// TIA Portal V20 export
// export: Created 2025-12-01T14:57:28.059015Z, ExportSetting None, DisplayName Totally Integrated Automation Portal, DisplayVersion V20 Update 3, DisplayName TIA Portal Openness, DisplayVersion V20 Update 3, DisplayName TIA Portal Version Control Interface, DisplayVersion V20 Update 3, DisplayName STEP 7 Professional, DisplayVersion V20 Update 3, DisplayName STEP 7 Safety, DisplayVersion V20 Update 2, DisplayName WinCC Basic/Comfort/Advanced, DisplayVersion V20 Update 3, DisplayName WinCC Professional, DisplayVersion V20 Update 3, DisplayName WinCC Unified, DisplayVersion V20 Update 3
FUNCTION_BLOCK "FB601_EntradaFija_Quimarox"   // FB601, LAD
{ S7_Optimized_Access := 'FALSE' }
// stored: AutoNumber false, SetENOAutomatically false
   VAR_INPUT
      MesaAnterior : UInt;
      MesaDeCarga : UInt;
      ID_Quimarox : UInt;
      ID_Elemento : UInt;
      EnTension : Bool;
      Termico : Bool;
      pHs_PosicionCarga : Bool;
      pHs_Protrusion : Bool;
      PRV_AVTF : Bool;
      PRV_DescargaActiva : Bool;
      V_FILTRO_pHsPresencia : Int;
      Pto_Ajuste_1 : Int;
   END_VAR
   VAR_OUTPUT
      PRV_PTF : Bool;   // permiso mesa anterior y avance de la siguiente
      PRV_FTF : Bool;
      PararElevador : Bool;
      ElevadorEnLenta : Bool;
      Avance_EntradaFija : Bool;
   END_VAR
   VAR_IN_OUT
      ROUTING_Destino : UInt;
      ROUTING_Etiqueta : UDInt;
   END_VAR
   VAR
      TMP_EnTension { S7_SetPoint := 'True'} : "FB910_CNT_UHS";
      FILTRO_pHsPresencia { S7_SetPoint := 'True'} : "FB910_CNT_UHS";
      EstadoAsociadoEnMesa : UInt;
      Aux_PeineDeCarga : UInt;
      PresenciaEnReset : Bool;
   END_VAR
   VAR_TEMP
      TMP_PeineDeCarga : UInt;
      TMP_PeineLiberar : UInt;
      MesaQuimarox : UInt;
      VagonReservado : UInt;
      NumeroUT : UInt;
      EsMesaTL : Bool;
      FILTRO_PosicionCarga : Bool;
   END_VAR
BEGIN

NETWORK
TITLE = ERROR - Rearme
/////////////////////////////////////////////////////////////
/////////////////////////////////////////////////////////////
/////////////////////////////////////////////////////////////
// Rearne de Errores
      SET;
      A     "DB902_Estado_ZonaMesa".EstadoMesas[#MesaDeCarga].Rearme_CBx;
      O     "DB902_Estado_ZonaMesa".EstadoMesas[#MesaDeCarga].PerReset_CBx;
      R     "DB900_Estado_Mesas".EstadoVI[#MesaDeCarga].Error_Mx;
      R     "DB900_Estado_Mesas".EstadoVI[#MesaDeCarga].Err_Protusion;
      R     "DB900_Estado_Mesas".EstadoVI[#MesaDeCarga].Err_TOut_Avance_E1_E3;
      R     "DB900_Estado_Mesas".EstadoVI[#MesaDeCarga].Err_DatosPLC;
      R     "DB900_Estado_Mesas".EstadoVI[#MesaDeCarga].Err_Termico_E1_E3;



NETWORK
TITLE = RECEP OK DE LA ORDEN -- NO SE UTILIZA
/////////////////////////////////////////////////////////////
/////////////////////////////////////////////////////////////
/////////////////////////////////////////////////////////////
// RECEP OK DE LA ORDEN
      SET;
      AN    "DB841_Recepcion".Mesa[#MesaDeCarga].Protocolo.Ord_S00;
      AN    "DB841_Recepcion".Mesa[#MesaDeCarga].Protocolo.Ord_S01;
      AN    "DB841_Recepcion".Mesa[#MesaDeCarga].Protocolo.Ord_S02;
      AN    "DB841_Recepcion".Mesa[#MesaDeCarga].Protocolo.Ord_S03;
      NOT;
      =     "DB840_Emision".Mesa[#MesaDeCarga].Protocolo.RecepOK;



NETWORK
TITLE = HMI - Manual
/////////////////////////////////////////////////////////////
/////////////////////////////////////////////////////////////
/////////////////////////////////////////////////////////////
// Para HMI >>> Manual
      SET;
      O     "DB902_Estado_ZonaMesa".EstadoMesas[#MesaDeCarga].Manual_CBx;
      =     "DB900_Estado_Mesas".EstadoVI[#MesaDeCarga].Manual;



NETWORK
TITLE = HMI - Entradas y Salidas de la Mesa
/////////////////////////////////////////////////////////////
/////////////////////////////////////////////////////////////
/////////////////////////////////////////////////////////////
// Entradas
      SET;
      A     #pHs_PosicionCarga;
      =     "DB900_Estado_Mesas".EstadoVI[#MesaDeCarga].En_PHS_1;
      SET;
      A     #pHs_Protrusion;
      =     "DB900_Estado_Mesas".EstadoVI[#MesaDeCarga].En_pHs_Prot1;

      SET;
      A     #Termico;
      =     "DB900_Estado_Mesas".EstadoVI[#MesaDeCarga].En_Termico1;

// Salidas
      SET;
      A     #Avance_EntradaFija;
      =     "DB900_Estado_Mesas".EstadoVI[#MesaDeCarga].Sa_Rod_Avance;



NETWORK
TITLE = Comprobacion de que la MESA es de TRACKING
/////////////////////////////////////////////////////////////
/////////////////////////////////////////////////////////////
/////////////////////////////////////////////////////////////
// Comprobar si es una Mesa de Tracking o Routing
      SET;
      A     "DB850_DefinicionMesas".Mesa[#MesaDeCarga].ConfigMesa.MesaTL;
      =     #EsMesaTL;



REGION Network 6: TMP - Espera En Tension
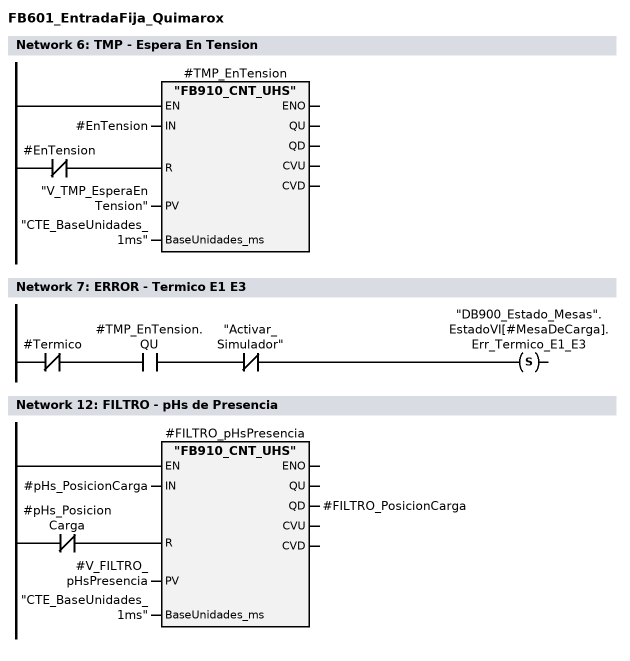
   RUNG wire#powerrail
      #TMP_EnTension(R := wire#w1, IN := #EnTension, PV := "V_TMP_EsperaEnTension", BaseUnidades_ms := "CTE_BaseUnidades_1ms", QU =>, QD =>, CVU =>, CVD =>)
   END_RUNG
   RUNG wire#powerrail
      I_Contact( #EnTension )
   END_RUNG wire#w1
   // the same network as SCL:
   #TMP_EnTension(IN := #EnTension,   // "FB910_CNT_UHS"
                  R := NOT #EnTension,
                  PV := "V_TMP_EsperaEnTension",
                  BaseUnidades_ms := "CTE_BaseUnidades_1ms");
END_REGION

REGION Network 7: ERROR - Termico E1 E3
   RUNG wire#powerrail
      I_Contact( #Termico )
      Contact( #TMP_EnTension.QU )
      I_Contact( "Activar_Simulador" )
      S_Coil( "DB900_Estado_Mesas".EstadoVI[#MesaDeCarga].Err_Termico_E1_E3 )
   END_RUNG
   // the same network as SCL:
   IF NOT #Termico AND #TMP_EnTension.QU AND NOT "Activar_Simulador" THEN
       "DB900_Estado_Mesas".EstadoVI[#MesaDeCarga].Err_Termico_E1_E3 := TRUE;
   END_IF;
END_REGION

NETWORK
TITLE = INICIALIZACION Previa
/////////////////////////////////////////////////////////////
/////////////////////////////////////////////////////////////
/////////////////////////////////////////////////////////////
      CLR;
      =     #PRV_PTF;
      =     #PRV_FTF;

      CLR;
      =     #ElevadorEnLenta;
      =     #PararElevador;
      =     #Avance_EntradaFija;

      CLR;
      =     "DB900_Estado_Mesas".EstadoVI[#MesaDeCarga].Etapas_Reset;
      =     "DB900_Estado_Mesas".EstadoVI[#MesaDeCarga].Etapa_Vacia;
      =     "DB900_Estado_Mesas".EstadoVI[#MesaDeCarga].Etapa_Cargada;
      =     "DB900_Estado_Mesas".EstadoVI[#MesaDeCarga].Etapas_Carga_E1;
      =     "DB900_Estado_Mesas".EstadoVI[#MesaDeCarga].Etapas_Descarga_S0;



NETWORK
TITLE = SISTEMA - Paro Blando
/////////////////////////////////////////////////////////////
/////////////////////////////////////////////////////////////
/////////////////////////////////////////////////////////////
// - Inicializar Variables de PARO BLANDO
      CLR;
      =     "DB900_Estado_Mesas".EstadoVI[#MesaDeCarga].Paro_Blando;

/////////////////////////////////////////////////////////////
// - Existe PARO BLANDO ???
      SET;
      AN    "DB902_Estado_ZonaMesa".EstadoMesas[#MesaDeCarga].ParoBlando_CBx;
      JC    NoRealizandose_ParoBlando;

/////////////////////////////////////////////////////////////
// - Fin de PARO BLANDO
      SET;
      =     "DB900_Estado_Mesas".EstadoVI[#MesaDeCarga].Paro_Blando;


/////////////////////////////////////////////////////////////
/////////////////////////////////////////////////////////////
/////////////////////////////////////////////////////////////
// - Final Tratamiento del PARO BLANDO
NoRealizandose_ParoBlando:NOP   0;



NETWORK
TITLE = SISTEMA - Reset
/////////////////////////////////////////////////////////////
/////////////////////////////////////////////////////////////
/////////////////////////////////////////////////////////////
// -- Inicializar Variables de RESET
      SET;
      AN    "DB902_Estado_ZonaMesa".EstadoMesas[#MesaDeCarga].PerReset_CBx;
      R     "DB900_Estado_Mesas".EstadoVI[#MesaDeCarga].Fin_VI;
      R     #PresenciaEnReset;

/////////////////////////////////////////////////////////////
/////////////////////////////////////////////////////////////
/////////////////////////////////////////////////////////////
// - Existe RESET ??
      SET;
      AN    "DB902_Estado_ZonaMesa".EstadoMesas[#MesaDeCarga].PerReset_CBx;
      JC    NoRealizandose_Reset;

      L     0;  // Estado de La Mesa = 0
      T     #EstadoAsociadoEnMesa;
      SET;
      =     "DB900_Estado_Mesas".EstadoVI[#MesaDeCarga].Etapas_Reset;

/////////////////////////////////////////////////////////////
/////////////////////////////////////////////////////////////
/////////////////////////////////////////////////////////////
// - Emision de Presencia en caso de Reset
      SET;  // Presencia >>> Reset Total
      A     #pHs_PosicionCarga;
      A     "DB831_Mesas".Mesas[#MesaDeCarga].Memorias.M_ResetTotal;
      AN    #PresenciaEnReset;
      JC    Enviar_PresenciaEnResetTotal;

      SET;  // Presencia >>> Reset Parcial
      A     #pHs_PosicionCarga;
      A     "DB831_Mesas".Mesas[#MesaDeCarga].Memorias.M_ResetParcial;
      AN    #PresenciaEnReset;
      JC    Enviar_PresenciaEnResetParcial;

      JU    Final_PresenciaEnReset;

// - Presencia en Reset TOTAL >>> Enviar NUUT
Enviar_PresenciaEnResetTotal:NOP   0;
      CALL  "FC723_InsertarUT_EnMesa"
      ( MesaActual := #MesaDeCarga,
        NumeroUT   := #NumeroUT
      );
      L     132;  // Envio de Nueva UT en RESET
      T     "DB812_UTs_Control".UT[#NumeroUT].EstadoEventoAGenerar;

      SET;  // Ya esta Avisado el JdT
      S     #PresenciaEnReset;

      JU    Final_PresenciaEnReset;

// - Presencia en Reset Parcial >>> Enviar LOCA en Reset Pantalla
Enviar_PresenciaEnResetParcial:NOP   0;
      L     "DB810_ColasMesas".Colas[#MesaDeCarga].UT_PrimeraMesa;
      T     #NumeroUT;

      L     #NumeroUT;  // Comprobar que Existe UT
      L     0;
      ==I;
      JC    ErrorDatosCargada;

      L     101;  // Envio de LOCA en RESET
      T     "DB812_UTs_Control".UT[#NumeroUT].EstadoEventoAGenerar;

      SET;  // Ya esta Avisado el JdT
      S     #PresenciaEnReset;

      JU    Final_PresenciaEnReset;

// - Final de la Presencia En Reset
Final_PresenciaEnReset:NOP   0;


/////////////////////////////////////////////////////////////
/////////////////////////////////////////////////////////////
/////////////////////////////////////////////////////////////
// - Fin de RESET
      SET;  // Con Presencia de Carga >>> TOTAL
      A(;
      L     "DB810_ColasMesas".Colas[#MesaDeCarga].UT_PrimeraMesa;
      L     0;
      ==I;
      );
      A     #pHs_PosicionCarga;
      A     #PresenciaEnReset;
      A     "DB831_Mesas".Mesas[#MesaDeCarga].Memorias.M_ResetTotal;
      S     "DB900_Estado_Mesas".EstadoVI[#MesaDeCarga].Fin_VI;

      SET;  // Con Presencia de Carga >>> PARCIAL
      A     #pHs_PosicionCarga;
      A     #PresenciaEnReset;
      A     "DB831_Mesas".Mesas[#MesaDeCarga].Memorias.M_ResetParcial;
      S     "DB900_Estado_Mesas".EstadoVI[#MesaDeCarga].Fin_VI;


      SET;  // Sin Presencia de Carga
      AN    #pHs_PosicionCarga;
      S     "DB900_Estado_Mesas".EstadoVI[#MesaDeCarga].Fin_VI;

      BE;

/////////////////////////////////////////////////////////////
/////////////////////////////////////////////////////////////
/////////////////////////////////////////////////////////////
// - Final Tratamiento del RESET
NoRealizandose_Reset:NOP   0;



NETWORK
TITLE = >>>>>>>>>>>>>>>>>>>>>>>>>>>>>>>>>>>>>>>>>>>>>>>>>>>>>>>>>>>>>>>>>>>

REGION Network 12: FILTRO - pHs de Presencia
   RUNG wire#powerrail
      #FILTRO_pHsPresencia(R := wire#w1, IN := #pHs_PosicionCarga, PV := #V_FILTRO_pHsPresencia, BaseUnidades_ms := "CTE_BaseUnidades_1ms", QU =>, QD => #FILTRO_PosicionCarga, CVU =>, CVD =>)
   END_RUNG
   RUNG wire#powerrail
      I_Contact( #pHs_PosicionCarga )
   END_RUNG wire#w1
   // the same network as SCL:
   #FILTRO_pHsPresencia(IN := #pHs_PosicionCarga,   // "FB910_CNT_UHS"
                        R := NOT #pHs_PosicionCarga,
                        PV := #V_FILTRO_pHsPresencia,
                        BaseUnidades_ms := "CTE_BaseUnidades_1ms",
                        QD => #FILTRO_PosicionCarga);
END_REGION

NETWORK
TITLE = >>>>>>>>>>>>>>>>>>>>>>>>>>>>>>>>>>>>>>>>>>>>>>>>>>>>>>>>>>>>>>>>>>>

NETWORK
TITLE = DISTRIBUCION >>> Control Etapa Activa
/////////////////////////////////////////////////////////////////////////////////////
/////////////////////////////////////////////////////////////////////////////////////
/////////////////////////////////////////////////////////////////////////////////////
// -- Listado de saltos de programa  >>> Estado
      L     #EstadoAsociadoEnMesa;
      JL    ESTADO_PorDefecto;

      JU    ETAPA_00_EnReset;  // En Reset
      JU    ETAPA_01_EnReposo;  // En Reposo
      JU    ETAPA_02_PrevioCarga_ComprobarRuta;  // Previo Carga >>> Comprobar Ruta
      JU    Etapa_03_PrevioCarga_ReservaPeine;  // Previo Carga >>>Gestion reserva del peine
      JU    ETAPA_04_PrevioCarga_Sincroniza;  // Previo Carga >>> espera sincronizacion con peine
      JU    ETAPA_05_Cargando;  // Cargando >>> Entrada
      JU    Etapa_06_FinDeCarga;  // Fin de la Carga
      JU    Etapa_07_CargaDelPeine;  // Fin de la Carga del Peine

ESTADO_PorDefecto:JU    FinFuncion;



NETWORK
TITLE = ETAPA 00 >>> En Reset
/////////////////////////////////////////////////////////////////////////////////////
/////////////////////////////////////////////////////////////////////////////////////
/////////////////////////////////////////////////////////////////////////////////////
ETAPA_00_EnReset:NOP   0;
      SET;
      =     "DB900_Estado_Mesas".EstadoVI[#MesaDeCarga].Etapas_Reset;


/////////////////////////////////////////////////////////////////////////////////////
// generación de error de protusion
      SET;
      AN    #pHs_Protrusion;
      JC    ErrorProtrusion;


/////////////////////////////////////////////////////////////////////////////////////
// Tiene que estar en Marcha y Sin Error para continuar
      SET;
      AN    "DB902_Estado_ZonaMesa".EstadoMesas[#MesaDeCarga].Marcha_CBx;
      O     "DB902_Estado_ZonaMesa".EstadoMesas[#MesaDeCarga].Error_CBx;
      JC    ET00_PararElevador;


/////////////////////////////////////////////////////////////////////////////////////
// Vacio >>> Sin Aviso de Carga
      SET;
      AN    #FILTRO_PosicionCarga;
      AN    #PRV_AVTF;
      JC    ET00_IrEtapa_01_EnReposo;

// Vacio >>> Con Aviso de Carga
      SET;
      AN    #FILTRO_PosicionCarga;
      A     #PRV_AVTF;
      JC    ET00_IrEtapa_02_PrevioCarga;

// Con Carga
      SET;
      A     #FILTRO_PosicionCarga;
      JC    ET00_IrEtapa_07_CargaDelPeine;
      BE;


/////////////////////////////////////////////////////////////////////////////////////
/////////////////////////////////////////////////////////////////////////////////////
/////////////////////////////////////////////////////////////////////////////////////
ET00_PararElevador:NOP   0;
      SET;
      =     #PararElevador;
      BE;


/////////////////////////////////////////////////////////////////////////////////////
/////////////////////////////////////////////////////////////////////////////////////
/////////////////////////////////////////////////////////////////////////////////////
ET00_IrEtapa_01_EnReposo:NOP   0;
      L     1;
      T     #EstadoAsociadoEnMesa;
      JU    ETAPA_01_EnReposo;


/////////////////////////////////////////////////////////////////////////////////////
/////////////////////////////////////////////////////////////////////////////////////
/////////////////////////////////////////////////////////////////////////////////////
ET00_IrEtapa_02_PrevioCarga:NOP   0;
      L     2;
      T     #EstadoAsociadoEnMesa;
      JU    ETAPA_02_PrevioCarga_ComprobarRuta;


/////////////////////////////////////////////////////////////////////////////////////
/////////////////////////////////////////////////////////////////////////////////////
/////////////////////////////////////////////////////////////////////////////////////
ET00_IrEtapa_07_CargaDelPeine:NOP   0;
      SET;  // No existe UT >>> Error de Datos
      A(;
      L     "DB810_ColasMesas".Colas[#MesaDeCarga].UT_PrimeraMesa;
      L     0;
      ==I;
      );
      AN    #EsMesaTL;
      JC    ErrorDatosCargada;

      L     7;
      T     #EstadoAsociadoEnMesa;
      JU    Etapa_07_CargaDelPeine;



NETWORK
TITLE = ETAPA 01 >>> En Reposo
/////////////////////////////////////////////////////////////////////////////////////
/////////////////////////////////////////////////////////////////////////////////////
/////////////////////////////////////////////////////////////////////////////////////
ETAPA_01_EnReposo:NOP   0;
      SET;
      =     "DB900_Estado_Mesas".EstadoVI[#MesaDeCarga].Etapa_Vacia;


/////////////////////////////////////////////////////////////////////////////////////
// generación de error de protusion cuando la mesa está vacía
      SET;
      AN    #pHs_Protrusion;
      JC    ErrorProtrusion;

/////////////////////////////////////////////////////////////////////////////////////
/////////////////////////////////////////////////////////////////////////////////////
/////////////////////////////////////////////////////////////////////////////////////
// Si Viene un Peine >>> Reservado para el Elemento >>> LIBERAR Peine
      SET;  // --- Sin Ventana
      AN    "DB602_ElementosQuimarox".Quimarox[#ID_Quimarox].Elementos[#ID_Elemento].Hay_Carrier_en_ventana;
      JC    ET01_PorReserva_NoLiberarPeine;

      L     "DB602_ElementosQuimarox".Quimarox[#ID_Quimarox].Elementos[#ID_Elemento].Numero_carrier;
      T     #TMP_PeineLiberar;

      SET;  // --- Sin Reserva
      AN    "DB601_PeinesQuimarox".Quimarox[#ID_Quimarox].vagon[#TMP_PeineLiberar].vagon_reservado_carga;
      JC    ET01_PorReserva_NoLiberarPeine;

      SET;  // --- No es para el elemento
      L     "DB601_PeinesQuimarox".Quimarox[#ID_Quimarox].vagon[#TMP_PeineLiberar].punto_entrada_carga;
      L     #ID_Elemento;
      <>I;
      JC    ET01_PorReserva_NoLiberarPeine;

/////////////////////////////////////////////////////////////////////////////////////
      SET;  // --- Liberar Peine
      R     "DB601_PeinesQuimarox".Quimarox[#ID_Quimarox].vagon[#TMP_PeineLiberar].vagon_reservado_carga;

      L     0;
      T     "DB601_PeinesQuimarox".Quimarox[#ID_Quimarox].vagon[#TMP_PeineLiberar].punto_entrada_carga;

/////////////////////////////////////////////////////////////////////////////////////
ET01_PorReserva_NoLiberarPeine:NOP   0;



/////////////////////////////////////////////////////////////////////////////////////
/////////////////////////////////////////////////////////////////////////////////////
/////////////////////////////////////////////////////////////////////////////////////
// comprobar estado correcto de reposo
      SET;
      AN    #PRV_AVTF;
      AN    #FILTRO_PosicionCarga;
      A     #pHs_Protrusion;
      JC    FinFuncion;

/////////////////////////////////////////////////////////////////////////////////////
// condiciones para pasar a la etapa cargada
      SET;
      A     #PRV_AVTF;
      AN    #FILTRO_PosicionCarga;
      A     #pHs_Protrusion;
      JC    ET01_IrEtapa_02_PrevioCarga;

      BE;


/////////////////////////////////////////////////////////////////////////////////////
/////////////////////////////////////////////////////////////////////////////////////
/////////////////////////////////////////////////////////////////////////////////////
ET01_IrEtapa_02_PrevioCarga:NOP   0;
      L     2;  // tengo una caja, paso a extraer orden
      T     #EstadoAsociadoEnMesa;
      JU    ETAPA_02_PrevioCarga_ComprobarRuta;



NETWORK
TITLE = ETAPA 02 >>> Comprobar Ruta
/////////////////////////////////////////////////////////////////////////////////////
/////////////////////////////////////////////////////////////////////////////////////
/////////////////////////////////////////////////////////////////////////////////////
ETAPA_02_PrevioCarga_ComprobarRuta:NOP   0;
      SET;
      =     "DB900_Estado_Mesas".EstadoVI[#MesaDeCarga].Etapa_Vacia;


/////////////////////////////////////////////////////////////////////////////////////
// generación de error de protusion cuando la mesa está vacía
      SET;
      AN    #pHs_Protrusion;
      JC    ErrorProtrusion;

/////////////////////////////////////////////////////////////////////////////////////
/////////////////////////////////////////////////////////////////////////////////////
/////////////////////////////////////////////////////////////////////////////////////
/// --- Comprobacion del TIPO de MESA
      SET;
      AN    #EsMesaTL;
      JC    TRACKING_ComprobarRuta;
      JU    ROUTING_ComprobarRuta;

/////////////////////////////////////////////////////////////////////////////////////
/// --- Comprobacion de Ruta en una MESA de ROUTING
ROUTING_ComprobarRuta:NOP   0;
      L     #ROUTING_Destino;
      L     0;
      ==I;
      JC    FinFuncion;
      JU    FINAL_ComprobacionDeRuta;

/////////////////////////////////////////////////////////////////////////////////////
/// --- Comprobacion de Ruta en una MESA de TRACKING
TRACKING_ComprobarRuta:NOP   0;
      L     "DB810_ColasMesas".Colas[#MesaAnterior].UT_PrimeraMesa;
      T     #NumeroUT;

      SET;
      L     #NumeroUT;  // Debe existir UT
      L     0;
      ==I;
      JC    FinFuncion;

// si la mesa actual y la de destino es la misma, significa que aún no tenemos destino
// y tenemos que esperar
      SET;
      L     "DB812_UTs_Control".UT[#NumeroUT].MesaActual;
      L     "DB812_UTs_Control".UT[#NumeroUT].MesaDestino;
      ==I;
      JC    FinFuncion;

      SET;
      L     0;
      L     "DB812_UTs_Control".UT[#NumeroUT].MesaDestino;
      ==I;
      JC    FinFuncion;

      JU    FINAL_ComprobacionDeRuta;


/////////////////////////////////////////////////////////////////////////////////////
/////////////////////////////////////////////////////////////////////////////////////
/////////////////////////////////////////////////////////////////////////////////////
/// --- Final de la Comprobacion de Ruta
FINAL_ComprobacionDeRuta:NOP   0;
      L     3;
      T     #EstadoAsociadoEnMesa;
      JU    Etapa_03_PrevioCarga_ReservaPeine;



NETWORK
TITLE = ETAPA 03 >>> Reserva de Peine
/////////////////////////////////////////////////////////////////////////////////////
/////////////////////////////////////////////////////////////////////////////////////
/////////////////////////////////////////////////////////////////////////////////////
// Generación de la reserva del peine
Etapa_03_PrevioCarga_ReservaPeine:NOP   0;
      SET;
      =     "DB900_Estado_Mesas".EstadoVI[#MesaDeCarga].Etapa_Vacia;


/////////////////////////////////////////////////////////////////////////////////////
// revisamos error de protusion
      SET;
      AN    #pHs_Protrusion;
      JC    ErrorProtrusion;

/////////////////////////////////////////////////////////////////////////////////////
// rearme del error si ha desaparecido la caja   OJO!!!!!!!CAMBIADO
      SET;
      AN    #PRV_AVTF;
      AN    #FILTRO_PosicionCarga;
      A     #pHs_Protrusion;
      A     "DB902_Estado_ZonaMesa".EstadoMesas[#MesaDeCarga].Rearme_CBx;
      JC    ET03_IrEtapa_01_EnReposo;

/////////////////////////////////////////////////////////////////////////////////////
// generar reserva de peine >>> Mesa Fija (1)
      CALL  "FC602_ReservaPeine"
      ( ID_Quimarox          := #ID_Quimarox,
        ID_ElementoPeticion  := #ID_Elemento,
        TipoDeElemento       := 1,
        NumeroPeineReservado := #VagonReservado
      );

/////////////////////////////////////////////////////////////////////////////////////
// si el vagón reservado es cero, es que no se ha podido gestionar la reserva y nos quedamos a la espera
      SET;
      L     #VagonReservado;
      L     0;
      ==I;
      JC    FinFuncion;

/////////////////////////////////////////////////////////////////////////////////////
// como ya hemos hecho la petición y nos han devuelto el peine de reserva, saltamos a la espera de la sincronización
// si hemos realizado correctamente la reserva, guardamos el dato y evolucionamos de etapa
      L     #VagonReservado;
      T     #Aux_PeineDeCarga;

      L     4;
      T     #EstadoAsociadoEnMesa;
      JU    ETAPA_04_PrevioCarga_Sincroniza;


/////////////////////////////////////////////////////////////////////////////////////
/////////////////////////////////////////////////////////////////////////////////////
/////////////////////////////////////////////////////////////////////////////////////
ET03_IrEtapa_01_EnReposo:NOP   0;
      L     1;
      T     #EstadoAsociadoEnMesa;
      JU    ETAPA_01_EnReposo;



NETWORK
TITLE = ETAPA 04 >>> Sincronizacion
/////////////////////////////////////////////////////////////////////////////////////
/////////////////////////////////////////////////////////////////////////////////////
/////////////////////////////////////////////////////////////////////////////////////
// a la espera de la sincronización con el peine reservado para nosotros
ETAPA_04_PrevioCarga_Sincroniza:NOP   0;
      SET;
      =     "DB900_Estado_Mesas".EstadoVI[#MesaDeCarga].Etapas_Carga_E1;


/////////////////////////////////////////////////////////////////////////////////////
// revisamos error de protusion
      SET;
      AN    #pHs_Protrusion;
      JC    ErrorProtrusion;

/////////////////////////////////////////////////////////////////////////////////////
// Esperamos la sincronización con el vagón con el que
      SET;
      A     "DB602_ElementosQuimarox".Quimarox[#ID_Quimarox].Elementos[#ID_Elemento].Hay_Carrier_en_ventana;
      A(;
      L     "DB602_ElementosQuimarox".Quimarox[#ID_Quimarox].Elementos[#ID_Elemento].Numero_carrier;  // #datos_elemento.Numero_carrier
      L     #Aux_PeineDeCarga;
      ==I;
      );
      JC    ET04_IrEtapa_05_Cargando;

/////////////////////////////////////////////////////////////////////////////////////
// si no se dan las condiciones de inicio de carga tenemos que seguir esperando
      BE;


/////////////////////////////////////////////////////////////////////////////////////
/////////////////////////////////////////////////////////////////////////////////////
/////////////////////////////////////////////////////////////////////////////////////
ET04_IrEtapa_05_Cargando:NOP   0;
      L     5;  // saltamos al inicio de proceso de carga
      T     #EstadoAsociadoEnMesa;
      JU    ETAPA_05_Cargando;



NETWORK
TITLE = ETAPA 05 >>> Cargando >>> Entrada
/////////////////////////////////////////////////////////////////////////////////////
/////////////////////////////////////////////////////////////////////////////////////
/////////////////////////////////////////////////////////////////////////////////////
ETAPA_05_Cargando:NOP   0;
      SET;
      =     "DB900_Estado_Mesas".EstadoVI[#MesaDeCarga].Etapas_Carga_E1;

      SET;
      =     #PRV_PTF;
      =     #Avance_EntradaFija;
      CLR;
      =     #PRV_FTF;


/////////////////////////////////////////////////////////////////////////////////////
// Se ha cargado correctamente y generamos los datos para el peine
      SET;
      A     #FILTRO_PosicionCarga;
      A     #PRV_AVTF;
      A     #pHs_Protrusion;
      JC    ET05_IrEtapa_06_FinDeCarga;


/////////////////////////////////////////////////////////////////////////////////////
// Aqui tenemos que vigilar que nos se nos está cerrado la ventana intentando cargar
// primero comprobamos que no tenemos ya la ventana cerrada, porque sino tenemos que parar el elevador
      SET;
      AN    "DB602_ElementosQuimarox".Quimarox[#ID_Quimarox].Elementos[#ID_Elemento].Hay_Carrier_en_ventana;  //#datos_elemento.Hay_Carrier_en_ventana
      A(;
      ON    #pHs_Protrusion;
      O     #FILTRO_PosicionCarga;
      );
      JC    ErrorEnCarga;

// Si pasamos de Largo la ventana hay quitar la reserva
      SET;
      AN    "DB602_ElementosQuimarox".Quimarox[#ID_Quimarox].Elementos[#ID_Elemento].Hay_Carrier_en_ventana;
//      UN    #Filtro_PoscionCarga
//      U     #pHs_Protrusion
//      UN    #PRV_AVTF
      JC    ET05_PasadoVagon_SinCargar;

// si seguimos teniendo el carrier en ventana, comprobamos cuanta ventana tenemos. llegados a un punto, pasaremos a lenta
      SET;
      L     "DB602_ElementosQuimarox".Quimarox[#ID_Quimarox].Elementos[#ID_Elemento].Avance_carrier;
      L     #Pto_Ajuste_1;
      >=I;
      JC    ET05_PararElevador;


/////////////////////////////////////////////////////////////////////////////////////
      BE;


/////////////////////////////////////////////////////////////////////////////////////
/////////////////////////////////////////////////////////////////////////////////////
/////////////////////////////////////////////////////////////////////////////////////
ET05_VelocidadLenta:NOP   0;
      SET;
      =     #ElevadorEnLenta;
      BE;

/////////////////////////////////////////////////////////////////////////////////////
/////////////////////////////////////////////////////////////////////////////////////
/////////////////////////////////////////////////////////////////////////////////////
ET05_PararElevador:NOP   0;
      SET;
      =     #PararElevador;
      BE;

/////////////////////////////////////////////////////////////////////////////////////
/////////////////////////////////////////////////////////////////////////////////////
/////////////////////////////////////////////////////////////////////////////////////
ET05_PasadoVagon_SinCargar:NOP   0;
      CLR;
      =     #ElevadorEnLenta;
      =     #PRV_PTF;
      =     #Avance_EntradaFija;

      CLR;
      =     "DB601_PeinesQuimarox".Quimarox[#ID_Quimarox].vagon[#Aux_PeineDeCarga].vagon_reservado_carga;  //#datos_peine_tmp.vagon_reservado_carga
      L     0;
      T     "DB601_PeinesQuimarox".Quimarox[#ID_Quimarox].vagon[#Aux_PeineDeCarga].punto_entrada_carga;
      T     #Aux_PeineDeCarga;

      L     1;
      T     #EstadoAsociadoEnMesa;
      JU    ETAPA_01_EnReposo;


/////////////////////////////////////////////////////////////////////////////////////
/////////////////////////////////////////////////////////////////////////////////////
/////////////////////////////////////////////////////////////////////////////////////
ET05_IrEtapa_06_FinDeCarga:NOP   0;
      L     6;
      T     #EstadoAsociadoEnMesa;


/////////////////////////////////////////////////////////////////////////////////////
// - Comprobacion del TIPO de MESA
      SET;
      A     #EsMesaTL;
      JC    Etapa_06_FinDeCarga;

// - Traer la UT de la Mesa Anterior
      L     "DB810_ColasMesas".Colas[#MesaAnterior].UT_PrimeraMesa;
      T     #NumeroUT;

      SET;  // No existe UT >>> Error de Datos
      L     #NumeroUT;
      L     0;
      ==I;
      JC    ErrorDatosCargada;

      CALL  "FC724_CambiarUT_DeMesa"
      ( NumeroUT    := #NumeroUT,
        NuevaMesa   := #MesaDeCarga,
        AlPrincipio := "DB850_DefinicionMesas".Mesa[#MesaDeCarga].ConfigMesa.MeterAlPrincipio
      );  // Cambia la UT a la Nueva Mesa

      L     0;  // Es de Ordenes Especiales - Resetear
      T     "DB812_UTs_Control".UT[#NumeroUT].EstadoRecepcionUT;
      T     "DB812_UTs_Control".UT[#NumeroUT].EstadoEventoRecibido;
      T     "DB812_UTs_Control".UT[#NumeroUT].EstadoEmisionUT;
      L     100;  // Emitir evento LOCA
      T     "DB812_UTs_Control".UT[#NumeroUT].EstadoEventoAGenerar;

      JU    Etapa_06_FinDeCarga;



NETWORK
TITLE = ETAPA 06 >>> Fin de la Carga >>> Cargada
/////////////////////////////////////////////////////////////////////////////////////
/////////////////////////////////////////////////////////////////////////////////////
/////////////////////////////////////////////////////////////////////////////////////
Etapa_06_FinDeCarga:NOP   0;
      SET;
      =     "DB900_Estado_Mesas".EstadoVI[#MesaDeCarga].Etapas_Carga_E1;

      SET;
      =     #PRV_FTF;
      CLR;
      =     #PRV_PTF;
      =     #Avance_EntradaFija;


/////////////////////////////////////////////////////////////////////////////////////
// revisamos error de protusion
      SET;
      AN    #pHs_Protrusion;
      JC    ErrorProtrusion;

/////////////////////////////////////////////////////////////////////////////////////
// Cargado Correctamente
      SET;
      A     #FILTRO_PosicionCarga;
      A     #pHs_Protrusion;
      AN    #PRV_AVTF;
      AN    #PRV_DescargaActiva;
      JC    ET06_IrEtapa_07_CargaDelPeine;

      BE;


/////////////////////////////////////////////////////////////////////////////////////
/////////////////////////////////////////////////////////////////////////////////////
/////////////////////////////////////////////////////////////////////////////////////
ET06_IrEtapa_07_CargaDelPeine:NOP   0;
      L     7;
      T     #EstadoAsociadoEnMesa;
      JU    Etapa_07_CargaDelPeine;



NETWORK
TITLE = ETAPA 07 >>> Carga En Peine (Rellenar datos del Vagon)
/////////////////////////////////////////////////////////////////////////////////////
/////////////////////////////////////////////////////////////////////////////////////
/////////////////////////////////////////////////////////////////////////////////////
Etapa_07_CargaDelPeine:NOP   0;
      SET;
      =     "DB900_Estado_Mesas".EstadoVI[#MesaDeCarga].Etapas_Descarga_S0;


/////////////////////////////////////////////////////////////////////////////////////
      CLR;
      =     #PRV_PTF;
      =     #PRV_FTF;
      =     #Avance_EntradaFija;
      =     #ElevadorEnLenta;

      L     "DB602_ElementosQuimarox".Quimarox[#ID_Quimarox].Elementos[#ID_Elemento].Numero_carrier;
      T     #TMP_PeineDeCarga;  // Peine que esta pasando por el Elemento


/////////////////////////////////////////////////////////////////////////////////////
// revisamos error de protusion
      SET;
      AN    #pHs_Protrusion;
      JC    ErrorProtrusion;

/////////////////////////////////////////////////////////////////////////////////////
// Cargado Correctamente en el PEINE
      SET;
      AN    #FILTRO_PosicionCarga;
      A     #pHs_Protrusion;
      JC    FINALIZADO_CargaDelPeine;

      BE;


/////////////////////////////////////////////////////////////////////////////////////
/////////////////////////////////////////////////////////////////////////////////////
/////////////////////////////////////////////////////////////////////////////////////
// cargamos los datos de la UT al peine   >>>>> DEPENDIENDO DE TIPO DE DATOS
FINALIZADO_CargaDelPeine:NOP   0;

// Numero de Peine que lo ha recogido  ?????? CUIDADO
      L     #TMP_PeineDeCarga;
      T     #Aux_PeineDeCarga;

// Tipo de Mesa ROUTING o TRACKING
      SET;
      =     "DB601_PeinesQuimarox".Quimarox[#ID_Quimarox].vagon[#Aux_PeineDeCarga].Carrier_Cargado;  //#datos_peine_tmp.Carrier_Cargado

      SET;
      AN    #EsMesaTL;
      JC    TRACKING_PasoDeDatos;
      JU    ROUTING_PasoDeDatos;

/////////////////////////////////////////////////////////////////////////////////////
// --- DATOS DE ROUTING
ROUTING_PasoDeDatos:NOP   0;
      L     0;
      T     "DB601_PeinesQuimarox".Quimarox[#ID_Quimarox].vagon[#Aux_PeineDeCarga].DatosCarga.Mckey;
      L     #MesaDeCarga;
      T     "DB601_PeinesQuimarox".Quimarox[#ID_Quimarox].vagon[#Aux_PeineDeCarga].DatosCarga.MesaOrigen;
      L     #ROUTING_Destino;
      T     "DB601_PeinesQuimarox".Quimarox[#ID_Quimarox].vagon[#Aux_PeineDeCarga].DatosCarga.MesaDestino;
      T     "DB601_PeinesQuimarox".Quimarox[#ID_Quimarox].vagon[#Aux_PeineDeCarga].Destino_principal;

      L     #ROUTING_Etiqueta;
      T     "DB601_PeinesQuimarox".Quimarox[#ID_Quimarox].vagon[#Aux_PeineDeCarga].DatosCarga.EtiquetaRouter;

      L     "CTE_Evento_QCAR";
      T     "DB601_PeinesQuimarox".Quimarox[#ID_Quimarox].vagon[#Aux_PeineDeCarga].EventoAGenerar;

      L     0;
      T     #ROUTING_Destino;
      T     #ROUTING_Etiqueta;

      JU    FINAL_PasoDeDatos;

/////////////////////////////////////////////////////////////////////////////////////
// --- DATOS DE TRACKING
TRACKING_PasoDeDatos:NOP   0;
      L     "DB810_ColasMesas".Colas[#MesaDeCarga].UT_PrimeraMesa;
      T     #NumeroUT;

      SET;  // No existe UT >>> Error de Datos
      L     #NumeroUT;
      L     0;
      ==I;
      JC    ErrorDatosCargada;

      L     "DB812_UTs_Control".UT[#NumeroUT].Mckey;
      T     "DB601_PeinesQuimarox".Quimarox[#ID_Quimarox].vagon[#Aux_PeineDeCarga].DatosCarga.Mckey;
      L     "DB812_UTs_Control".UT[#NumeroUT].MesaActual;
      T     "DB601_PeinesQuimarox".Quimarox[#ID_Quimarox].vagon[#Aux_PeineDeCarga].DatosCarga.MesaOrigen;
      L     "DB812_UTs_Control".UT[#NumeroUT].MesaDestino;
      T     "DB601_PeinesQuimarox".Quimarox[#ID_Quimarox].vagon[#Aux_PeineDeCarga].DatosCarga.MesaDestino;
      T     "DB601_PeinesQuimarox".Quimarox[#ID_Quimarox].vagon[#Aux_PeineDeCarga].Destino_principal;  // ?????

      L     "DB814_UTs_Etiqueta".UT[#NumeroUT].EtiquetaRouter;
      T     "DB601_PeinesQuimarox".Quimarox[#ID_Quimarox].vagon[#Aux_PeineDeCarga].DatosCarga.EtiquetaRouter;

      L     "CTE_Evento_QCAR";
      T     "DB601_PeinesQuimarox".Quimarox[#ID_Quimarox].vagon[#Aux_PeineDeCarga].EventoAGenerar;
      L     131;
      T     "DB812_UTs_Control".UT[#NumeroUT].EstadoEventoAGenerar;

// Borrar UT Sin Avisar al JDT >>>> OJO
      CALL  "FC722_EliminarUT_DeMesa"
      ( NumeroUT := #NumeroUT
      );

      JU    FINAL_PasoDeDatos;


/////////////////////////////////////////////////////////////////////////////////////
/////////////////////////////////////////////////////////////////////////////////////
/////////////////////////////////////////////////////////////////////////////////////
FINAL_PasoDeDatos:NOP   0;
      CLR;
      =     "DB601_PeinesQuimarox".Quimarox[#ID_Quimarox].vagon[#Aux_PeineDeCarga].vagon_reservado_carga;  //#datos_peine_tmp.vagon_reservado_carga

      L     0;
      T     "DB601_PeinesQuimarox".Quimarox[#ID_Quimarox].vagon[#Aux_PeineDeCarga].punto_entrada_carga;
      T     #Aux_PeineDeCarga;

      L     1;
      T     #EstadoAsociadoEnMesa;  // volvemos a la posicion de reposo
      BE;



NETWORK
TITLE = >>>>>>>>>>>>>>>>>>>>>>>>>>>>>>>>>>>>>>>>>>>>>>>>>>>>>>>>>>>>>>>>>>>

NETWORK
TITLE = ERRRORES DE LA MESA >>> Activacion
/////////////////////////////////////////////////////////////////////////////////////
/////////////////////////////////////////////////////////////////////////////////////
/////////////////////////////////////////////////////////////////////////////////////
ErrorProtrusion:SET;
      =     "DB900_Estado_Mesas".EstadoVI[#MesaDeCarga].Error_Mx;
      =     "DB900_Estado_Mesas".EstadoVI[#MesaDeCarga].Err_Protusion;
      =     #PararElevador;
      BE;


/////////////////////////////////////////////////////////////////////////////////////
/////////////////////////////////////////////////////////////////////////////////////
/////////////////////////////////////////////////////////////////////////////////////
ErrorEnCarga:NOP   0;  // error en la carga
      SET;
      =     "DB900_Estado_Mesas".EstadoVI[#MesaDeCarga].Error_Mx;
      =     "DB900_Estado_Mesas".EstadoVI[#MesaDeCarga].Err_TOut_Avance_E1_E3;
      =     #PararElevador;
      BE;

/////////////////////////////////////////////////////////////////////////////////////
/////////////////////////////////////////////////////////////////////////////////////
/////////////////////////////////////////////////////////////////////////////////////
ErrorDatosCargada:NOP   0;  // error en la carga
      SET;
      =     "DB900_Estado_Mesas".EstadoVI[#MesaDeCarga].Error_Mx;
      =     "DB900_Estado_Mesas".EstadoVI[#MesaDeCarga].Err_DatosPLC;
      =     #PararElevador;
      BE;


NETWORK
TITLE = FINAL DE LA FUNCION
/////////////////////////////////////////////////////////////////////////////////////
/////////////////////////////////////////////////////////////////////////////////////
/////////////////////////////////////////////////////////////////////////////////////
FinFuncion:BE;


END_FUNCTION_BLOCK
